Yaskawa INFORM job: R2_ROBOTCALIB_WIDE.JBI

/JOB
//NAME R2_ROBOTCALIB_WIDE
///FOLDERNAME INNE
//POS
///NPOS 8,8,0,0,0,0
///TOOL 0
///POSTYPE PULSE
///PULSE
C00000=79983,53738,65838,70288,29625,-35518
C00001=71939,76999,90357,76529,34055,-39626
C00002=79212,52853,62162,67598,30817,-34195
C00003=79901,54065,66206,70411,29658,-35589
C00004=79790,53929,65556,69894,29853,-35331
C00005=136222,2244,-6496,-22625,28923,10856
C00006=136346,4001,-29094,-16018,43002,7207
C00007=79766,54027,65670,69937,29861,-35354
BC00000=398161,156221,441640
BC00001=108,156223,423137
BC00002=35,156223,999028
BC00003=398191,156253,1014637
BC00004=398161,1308293,441640
BC00005=108,1308295,423137
BC00006=109,1308295,1072495
BC00007=398191,1308324,1014636
//INST
///DATE 2023/10/17 12:53
///ATTR SC,RW
///GROUP1 RB1,BS1
NOP
MOVJ C00000 BC00000 VJ=0.78 PL=0
MOVJ C00001 BC00001 VJ=0.78 PL=0
MOVJ C00002 BC00002 VJ=0.78 PL=0
MOVJ C00003 BC00003 VJ=0.78 PL=0
'COMMENT
MOVJ C00004 BC00004 VJ=0.78 PL=0
MOVJ C00005 BC00005 VJ=0.78 PL=0
MOVJ C00006 BC00006 VJ=0.78 PL=0
MOVJ C00007 BC00007 VJ=0.78 PL=0
END
